Staubli VAL3: setLastError.pgx

program setLastError(num x_nError)
begin

  //Header begin

  // Describe functionality and purpose
  //
  //Input parameters
  // type param1: description (role, possible values,...)
  // param1 description (continued)
  // param1 description (continued)
  // type param2: description (role, possible values,...)
  // type param3: description (role, possible values,...)
  // ...
  //
  //Output parameters
  // type param1: description (role, possible values,...)
  // type param2: description (role, possible values,...)
  // type param3: description (role, possible values,...)
  // ...
  //
  //Examples
  // call examples (for public programs mostly)
  //
  //History
  // Creation: DD-MM-YY - AUTHOR NAME
  // Modification: DD-MM-YY - AUTHOR NAME - Description of modification
  // description of modification (continued)
  // description of modification (continued)
  // Modification: DD-MM-YY - AUTHOR NAME - Description of modification
  //Header end

  nLastError=x_nError

end
